FUNCTION_BLOCK FB_Hmi_Button EXTENDS FB_Hmi_Led
VAR
	_rButton: REFERENCE TO S_Hmi_Button;

	_behaviour: E_Hmi_ButtonBehaviour;
	_value: BOOL;
	_led: BOOL;

	_initialized: BOOL;
END_VAR

IF _initialized THEN
	IF _behaviour = _behaviour.MomentaryOff THEN
		_value := TRUE;
	ELSIF _behaviour = _behaviour.MomentaryOn THEN
		_value := FALSE;
	END_IF

	IF _rButton.Click THEN
		CASE _behaviour OF
			E_Hmi_ButtonBehaviour.MomentaryOff:
				Reset();

			E_Hmi_ButtonBehaviour.MomentaryOn:
				Set();

			E_Hmi_ButtonBehaviour.Reset:
				Reset();

			E_Hmi_ButtonBehaviour.Set:
				Set();

			E_Hmi_ButtonBehaviour.Toggle:
				Toggle();
		END_CASE

		_rButton.Click := FALSE;
	END_IF
END_IF

PROPERTY PUBLIC Enabled : BOOL
GET
Enabled := _rButton.Enabled;
END_GET
SET
_rButton.Enabled := Enabled;
END_SET
END_PROPERTY

METHOD PUBLIC Initialize : BOOL
VAR_INPUT
	rButton: REFERENCE TO S_Hmi_Button;
	behaviour: E_Hmi_ButtonBehaviour;
END_VAR
END_METHOD

PROPERTY PUBLIC Led : BOOL
GET
Led := _led;
END_GET
SET
IF _rButton.Enabled THEN
	_led := Led;
END_IF
END_SET
END_PROPERTY

METHOD PUBLIC Reset : BOOL
IF _rButton.Enabled THEN
	_value := FALSE;
END_IF
END_METHOD

METHOD PUBLIC Set : BOOL
IF _rButton.Enabled THEN
	_value := TRUE;
END_IF
END_METHOD

METHOD PUBLIC Toggle : BOOL
IF _rButton.Enabled THEN
	_value := NOT _value;
END_IF
END_METHOD

PROPERTY PUBLIC Value : BOOL
GET
Value := _value;
END_GET
END_PROPERTY

END_FUNCTION_BLOCK

(* stored: Version 1.1.0.1, ProductVersion 3.1.4024.10
   POU FB_Hmi_Button: Id {a617f7ad-fb3b-4a46-851f-875681a96aba}, SpecialFunc None
   Property Enabled: Id {5b4cf018-ce66-4b92-8000-7260fe469dc8}
   Get Get: Id {5d03b13b-c11f-4989-ae9e-058c70ae72aa}
   Set Set: Id {2793329d-7047-48a2-9868-24a2d32378e8}
   Method Initialize: Id {e3910462-5f99-46e6-a6aa-9b16848dc198}
   Property Led: Id {2886d8f7-91ae-4509-a03a-8ce26d6320e8}
   Get Get: Id {d00133b7-c570-4520-9dd4-1cc0b8ddc711}
   Set Set: Id {5c47a612-d18b-42a3-903a-a9bc5688f5ac}
   Method Reset: Id {e5c166a3-5f3c-4eb9-b57a-708a2a6197b7}
   Method Set: Id {d110b873-8a6f-4d1f-b710-60c6a34d74e5}
   Method Toggle: Id {2e7dfe79-cc01-47d2-a514-773e8cd4ab1d}
   Property Value: Id {4699e93b-d29c-4866-a3a4-a35fe790999d}
   Get Get: Id {ba3d2ae5-2beb-480e-86ae-d9f4f4c013ab} *)
